(* CoDeSys 2.3 export: PLC_PRG.EXP *)

(* POU PLC_PRG, LD *)
PROGRAM PLC_PRG
VAR
	S1: BOOL;
	S3: BOOL;
	res: BOOL;
	S2: BOOL;
	S4: BOOL;
	C3: CTUD;
	W1: BOOL;
	C4: CTUD;
	Ruch_Lewo: BOOL;
	Ruch_Dol: BOOL;
	DUMMY: BOOL;
	M1:MAPA;
	Ruch_Gora: BOOL;
	T_Ani: TON;
	C_Ani: CTU;
	SR1: SR;
	Reset_SR1: BOOL;
	SR2: SR;
	Reset_SR2: BOOL;
	SR3: SR;
	Reset_SR3: BOOL;
	Reset_SR4: BOOL;
	SR4: SR;
	T_Ruch: TON;
END_VAR
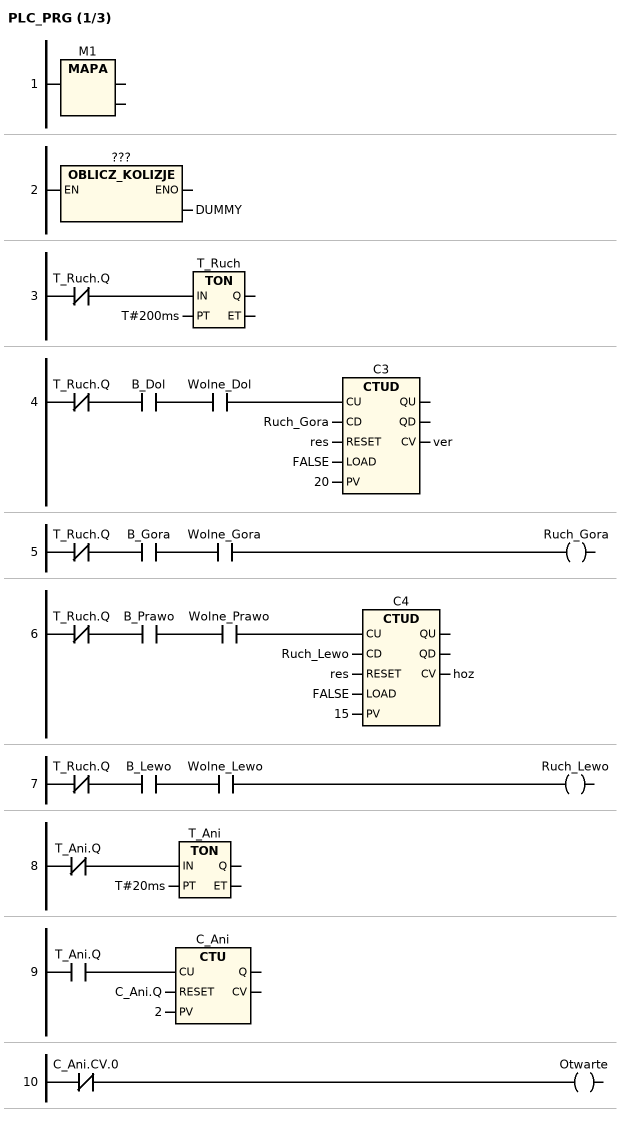
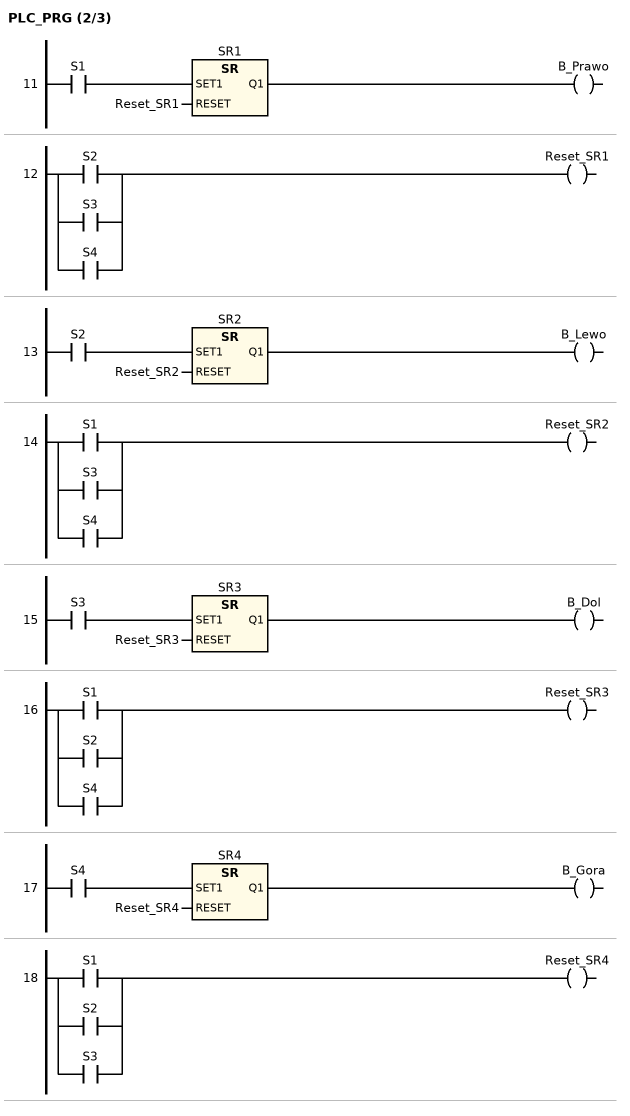
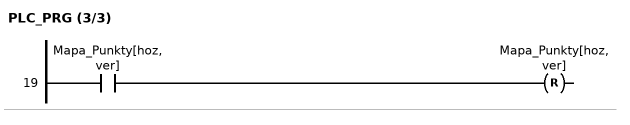
_LD_ (* Ladder Diagram *)
NETWORK 1
	M1:MAPA()
NETWORK 2
	*
		EN --- ???:OBLICZ_KOLIZJE() => DUMMY
NETWORK 3
	[/T_Ruch.Q] - T_Ruch:TON(IN: *, PT: T#200ms)
NETWORK 4
	[/T_Ruch.Q] - [B_Dol] - [Wolne_Dol] - C3:CTUD(CU: *, CD: Ruch_Gora, RESET: res, LOAD: FALSE, PV: 20, CV => ver)
NETWORK 5
	[/T_Ruch.Q] - [B_Gora] - [Wolne_Gora] --- (Ruch_Gora)
NETWORK 6
	[/T_Ruch.Q] - [B_Prawo] - [Wolne_Prawo] - C4:CTUD(CU: *, CD: Ruch_Lewo, RESET: res, LOAD: FALSE, PV: 15, CV => hoz)
NETWORK 7
	[/T_Ruch.Q] - [B_Lewo] - [Wolne_Lewo] --- (Ruch_Lewo)
NETWORK 8
	[/T_Ani.Q] - T_Ani:TON(IN: *, PT: T#20ms)
NETWORK 9
	[T_Ani.Q] - C_Ani:CTU(CU: *, RESET: C_Ani.Q, PV: 2)
NETWORK 10
	[/C_Ani.CV.0] --- (Otwarte)
NETWORK 11
	[S1] - SR1:SR(SET1: *, RESET: Reset_SR1) --- (B_Prawo)
NETWORK 12
	{ [S2] | [S3] | [S4] } --- (Reset_SR1)
NETWORK 13
	[S2] - SR2:SR(SET1: *, RESET: Reset_SR2) --- (B_Lewo)
NETWORK 14
	{ [S1] | [S3] | [S4] } --- (Reset_SR2)
NETWORK 15
	[S3] - SR3:SR(SET1: *, RESET: Reset_SR3) --- (B_Dol)
NETWORK 16
	{ [S1] | [S2] | [S4] } --- (Reset_SR3)
NETWORK 17
	[S4] - SR4:SR(SET1: *, RESET: Reset_SR4) --- (B_Gora)
NETWORK 18
	{ [S1] | [S2] | [S3] } --- (Reset_SR4)
NETWORK 19
	[Mapa_Punkty[hoz, ver]] --- (R Mapa_Punkty[hoz, ver])
_END_LD_
(* the same logic as Structured Text *)
(* Network 1 *)
M1();
(* Network 2: see the listing above *)
(* Network 3 *)
T_Ruch(IN := NOT T_Ruch.Q, PT := T#200ms);
(* Network 4 *)
C3(CU := NOT T_Ruch.Q AND B_Dol AND Wolne_Dol, CD := Ruch_Gora, RESET := res, LOAD := FALSE, PV := 20);
ver := C3.CV;
(* Network 5 *)
Ruch_Gora := NOT T_Ruch.Q AND B_Gora AND Wolne_Gora;
(* Network 6 *)
C4(CU := NOT T_Ruch.Q AND B_Prawo AND Wolne_Prawo, CD := Ruch_Lewo, RESET := res, LOAD := FALSE, PV := 15);
hoz := C4.CV;
(* Network 7 *)
Ruch_Lewo := NOT T_Ruch.Q AND B_Lewo AND Wolne_Lewo;
(* Network 8 *)
T_Ani(IN := NOT T_Ani.Q, PT := T#20ms);
(* Network 9 *)
C_Ani(CU := T_Ani.Q, RESET := C_Ani.Q, PV := 2);
(* Network 10 *)
Otwarte := NOT C_Ani.CV.0;
(* Network 11 *)
SR1(SET1 := S1, RESET := Reset_SR1);
B_Prawo := SR1.Q1;
(* Network 12 *)
Reset_SR1 := S2 OR S3 OR S4;
(* Network 13 *)
SR2(SET1 := S2, RESET := Reset_SR2);
B_Lewo := SR2.Q1;
(* Network 14 *)
Reset_SR2 := S1 OR S3 OR S4;
(* Network 15 *)
SR3(SET1 := S3, RESET := Reset_SR3);
B_Dol := SR3.Q1;
(* Network 16 *)
Reset_SR3 := S1 OR S2 OR S4;
(* Network 17 *)
SR4(SET1 := S4, RESET := Reset_SR4);
B_Gora := SR4.Q1;
(* Network 18 *)
Reset_SR4 := S1 OR S2 OR S3;
(* Network 19 *)
IF Mapa_Punkty[hoz, ver] THEN Mapa_Punkty[hoz, ver] := FALSE; END_IF;
END_PROGRAM
